{attribute 'GeneratedUsingTerminal: KL2652-0050'}
{attribute addProperty BoxType "KL2652-0050"}
{attribute addProperty Id "State_AutoAT %I*BOOL0State_RelayAT %I*BOOL0OutputAT %Q*BOOL0"}
{attribute addProperty CRC "1837855755"}
{attribute addProperty Size "0"}
TYPE Channel_6D8B740B :
STRUCT
	{attribute addProperty Name "State_Auto"}
	State_Auto AT %I* : BOOL;
	{attribute addProperty Name "State_Relay"}
	State_Relay AT %I* : BOOL;
	{attribute addProperty Name "Output"}
	Output AT %Q* : BOOL;
END_STRUCT
END_TYPE

(* stored: Version 1.2.0.0, ProductVersion 3.1.4024.9
   DUT Channel_6D8B740B: Id {ca6f1142-ea51-4d27-84d2-06d864e34d2d} *)
